// TIA Portal V17 export
// export: Created 2025-04-11T04:54:23.7658192Z, ExportSetting WithDefaults, DisplayName Totally Integrated Automation Portal, DisplayVersion V17, DisplayName TIA Portal Openness, DisplayVersion V17, DisplayName TIA Portal Version Control Interface, DisplayVersion V17, DisplayName SINAMICS Startdrive Advanced, DisplayVersion V17, DisplayName SINAMICS Startdrive G130, G150, S120, S150, SINAMICS MV, S210, DisplayVersion V17, DisplayName SINAMICS Startdrive G110M, G120, G120C, G120D, G120P, G115D, DisplayVersion V17, DisplayName STEP 7 Professional, DisplayVersion V17, DisplayName STEP 7 Safety, DisplayVersion V17, DisplayName WinCC Advanced, DisplayVersion V17
TYPE "UDT_Valve_Keep"
// stored: IsFailsafeCompliant false
   STRUCT
      IN_tOpenTime : Time := T#10S;   // 开阀超时时间
      IN_tCloseTime : Time := T#10S;   // 关阀超时时间
      IN_xALMEnable : Bool := TRUE;   // 报警使能
      INOUT_udiCount : UDInt;   // 计次
   END_STRUCT;
END_TYPE
